(* Logix 5000 project; controller EuniceF_ICA7 vendor 1 type 14 code 150 rev 37.11; software revision 37.00 *)

TASK MainTask (continuous, watchdog 500 ms) : MainProgram

MODULES
   Local : vendor 1 type 14 code 150 (Compact 0, rev 37.11)
      Discrete_IO : Embedded (Compact 1, rev 3.1, Output RPI 20 ms)
      Analog_IO : Embedded (Compact 2, rev 1.1, Output RPI 80 ms)
      Counters : Embedded (Compact 3, rev 1.1, Output RPI 20 ms)
END_MODULES

VAR_GLOBAL   (* controller tags *)
   BOTTOMLIM : ALIAS FOR Local:1:I.Data.1;
   CRUNCH : ALIAS FOR Local:1:I.Data.15;
   DOWN : ALIAS FOR Local:1:O.Data.1;
   GODOWN : ALIAS FOR Local:1:I.Data.12;
   GOUP : ALIAS FOR Local:1:I.Data.11;
   IHIH : BOOL;
   STOP : ALIAS FOR Local:1:I.Data.9;
   TOPLIM : ALIAS FOR Local:1:I.Data.0;
   UP : ALIAS FOR Local:1:O.Data.2;
END_VAR

PROGRAM MainProgram   (* main routine MainRoutine *)

ROUTINE MainRoutine   (* ladder *)
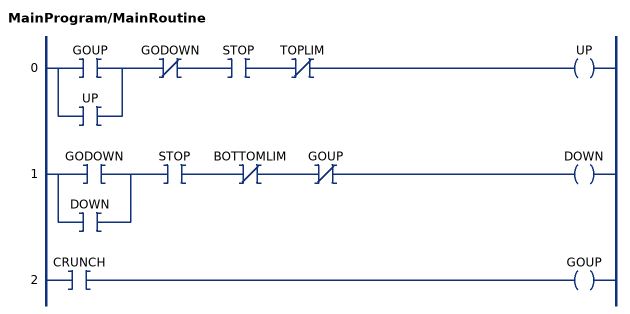
   0: [XIC(GOUP) ,XIC(UP) ]XIO(GODOWN)XIC(STOP)XIO(TOPLIM)OTE(UP);
   1: [XIC(GODOWN) ,XIC(DOWN) ]XIC(STOP)XIO(BOTTOMLIM)XIO(GOUP)OTE(DOWN);
   2: XIC(CRUNCH)OTE(GOUP);
END_ROUTINE
END_PROGRAM
